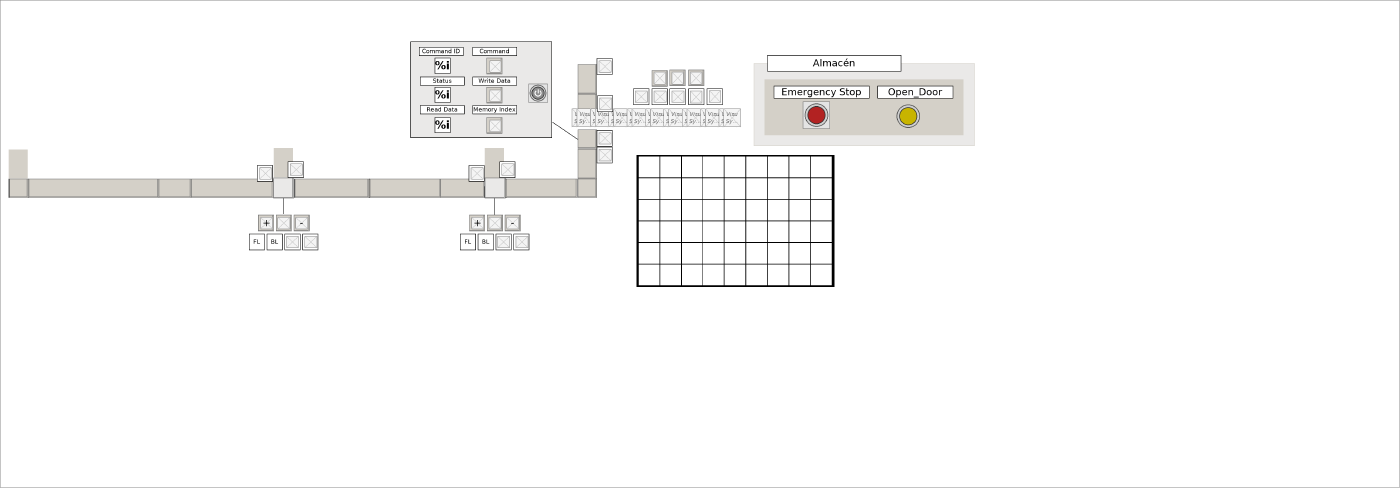
VISUALIZATION Linea_Almacen_Manual  // 2593x904
    Line (916,352) (916,399)
    Rectangle (889,284 55x35), angle 90
    Rectangle (155,228 35x241), angle 90
    Rectangle (984,282 35x132), angle 90
    Rectangle (306,318 35x60), angle 90
    Rectangle (412,272 35x152), angle 90
    Rectangle (506,329 38x38), angle 90
    Rectangle (597,280 35x137), angle 90
    Rectangle (732,283 35x131), angle 90
    Rectangle (839,308 35x81), angle 90
    Rectangle (906,336 21x38), angle 90
    Rectangle (17,331 35x35), angle 90
    Rectangle (8,286 53x35), angle 90
    Rectangle (498,284 54x35), angle 90
    Line (525,349) (525,396)
    InvisibleInput (1761,606 90x136)
    InvisibleInput (582,613 18x35)
    Button (17,331 35x35), colour toggle: GVL.Curved_Roller_Conveyor_1_CCW, pressed state: GVL.Curved_Roller_Conveyor_1_CCW
        OnMouseClick: toggle GVL.Curved_Roller_Conveyor_1_CCW
    Button (53,331 241x35), colour toggle: GVL.Roller_Conveyor_6m_1, pressed state: GVL.Roller_Conveyor_6m_1
        OnMouseClick: toggle GVL.Roller_Conveyor_6m_1
    Button (294,331 60x35), colour toggle: GVL.Chain_Transfer_1_mas, pressed state: GVL.Chain_Transfer_1_mas
        OnMouseClick: toggle GVL.Chain_Transfer_1_mas
    Button (354,331 152x35), colour toggle: GVL.Roller_Conveyor_4m_1, pressed state: GVL.Roller_Conveyor_4m_1
        OnMouseClick: toggle GVL.Roller_Conveyor_4m_1
    Button (506,329 38x38), pressed state: GVL.Roller_Conveyor_2m_2
    Button (546,331 137x35), colour toggle: GVL.Roller_Conveyor_6m_2, pressed state: GVL.Roller_Conveyor_6m_2
        OnMouseClick: toggle GVL.Roller_Conveyor_6m_2
    Button (685,331 131x35), colour toggle: GVL.Roller_Conveyor_4m_2, pressed state: GVL.Roller_Conveyor_4m_2
        OnMouseClick: toggle GVL.Roller_Conveyor_4m_2
    Button (816,331 81x35), colour toggle: GVL.Roller_Conveyor_2m_5, pressed state: GVL.Roller_Conveyor_2m_5
        OnMouseClick: toggle GVL.Roller_Conveyor_2m_5
    Button (898,329 38x38), colour toggle: GVL.Roller_Conveyor_2m_2, pressed state: GVL.Roller_Conveyor_2m_2
    Button (938,331 131x35), colour toggle: GVL.Roller_Conveyor_2m_2, pressed state: GVL.Roller_Conveyor_2m_2
        OnMouseClick: toggle GVL.Roller_Conveyor_2m_2
    Button (1070,331 35x35), colour toggle: GVL.Curved_Roller_Conveyor_2_CW, pressed state: GVL.Curved_Roller_Conveyor_2_CW
        OnMouseClick: toggle GVL.Curved_Roller_Conveyor_2_CW
    Button (1070,276 35x55), colour toggle: GVL.Roller_Conveyor_2m_8, pressed state: GVL.Roller_Conveyor_2m_8
        OnMouseClick: toggle GVL.Roller_Conveyor_2m_8
    Button (1070,240 35x35), colour toggle: GVL.Loading_Conveyor_1, pressed state: GVL.Loading_Conveyor_1
        OnMouseClick: toggle GVL.Loading_Conveyor_1
    Button (1070,174 35x35), colour toggle: GVL.Loading_Conveyor_2, pressed state: GVL.Loading_Conveyor_2
        OnMouseClick: toggle GVL.Loading_Conveyor_2
    Button (1070,119 35x55), colour toggle: GVL.Roller_Conveyor_2m_9, pressed state: GVL.Roller_Conveyor_2m_8
        OnMouseClick: toggle GVL.Roller_Conveyor_2m_9
    Rectangle (1179,287 366x244)
    Rectangle (1302,289 40x40)
    Rectangle (1302,329 40x40)
    Rectangle (1302,369 40x40)
    Rectangle (1302,409 40x40)
    Rectangle (1302,449 40x40)
    Rectangle (1302,489 40x40)
    Rectangle (1342,289 40x40)
    Rectangle (1342,329 40x40)
    Rectangle (1342,369 40x40)
    Rectangle (1342,409 40x40)
    Rectangle (1342,449 40x40)
    Rectangle (1342,489 40x40)
    Rectangle (1382,289 40x40)
    Rectangle (1382,329 40x40)
    Rectangle (1382,369 40x40)
    Rectangle (1382,409 40x40)
    Rectangle (1382,449 40x40)
    Rectangle (1382,489 40x40)
    Rectangle (1422,289 40x40)
    Rectangle (1422,329 40x40)
    Rectangle (1422,369 40x40)
    Rectangle (1422,409 40x40)
    Rectangle (1422,449 40x40)
    Rectangle (1422,489 40x40)
    Rectangle (1462,289 40x40)
    Rectangle (1462,329 40x40)
    Rectangle (1462,369 40x40)
    Rectangle (1462,409 40x40)
    Rectangle (1462,449 40x40)
    Rectangle (1462,489 40x40)
    Rectangle (1502,289 40x40)
    Rectangle (1502,329 40x40)
    Rectangle (1502,369 40x40)
    Rectangle (1502,409 40x40)
    Rectangle (1502,449 40x40)
    Rectangle (1502,489 40x40)
    Rectangle (1182,289 40x40)
    Rectangle (1182,329 40x40)
    Rectangle (1182,369 40x40)
    Rectangle (1182,409 40x40)
    Rectangle (1182,449 40x40)
    Rectangle (1182,489 40x40)
    Rectangle (1222,289 40x40)
    Rectangle (1222,329 40x40)
    Rectangle (1222,369 40x40)
    Rectangle (1222,409 40x40)
    Rectangle (1222,449 40x40)
    Rectangle (1222,489 40x40)
    Rectangle (1262,289 40x40)
    Rectangle (1262,329 40x40)
    Rectangle (1262,369 40x40)
    Rectangle (1262,409 40x40)
    Rectangle (1262,449 40x40)
    Rectangle (1262,489 40x40)
    Rectangle (1182,289 40x40), colour toggle: GVL.Clasificados[45].Visibilidad_Azul, invisible if: GVL.Clasificados[45].Visibilidad_Azul
    Rectangle (1182,329 40x40), colour toggle: GVL.Clasificados[36].Visibilidad_Azul, invisible if: GVL.Clasificados[36].Visibilidad_Azul
    Rectangle (1182,369 40x40), colour toggle: GVL.Clasificados[27].Visibilidad_Azul, invisible if: GVL.Clasificados[27].Visibilidad_Azul
    Rectangle (1182,409 40x40), colour toggle: GVL.Clasificados[18].Visibilidad_Azul, invisible if: GVL.Clasificados[18].Visibilidad_Azul
    Rectangle (1182,449 40x40), colour toggle: GVL.Clasificados[9].Visibilidad_Azul, invisible if: GVL.Clasificados[9].Visibilidad_Azul
    Rectangle (1182,489 40x40), colour toggle: GVL.Clasificados[0].Visibilidad_Azul, invisible if: GVL.Clasificados[0].Visibilidad_Azul
    Rectangle (1222,290 40x40)
    Rectangle (1222,330 40x40)
    Rectangle (1222,370 40x40)
    Rectangle (1222,410 40x40)
    Rectangle (1222,450 40x40)
    Rectangle (1222,490 40x40)
    Rectangle (1222,289 40x40), colour toggle: GVL.Clasificados[46].Visibilidad_Azul, invisible if: GVL.Clasificados[46].Visibilidad_Azul
    Rectangle (1222,329 40x40), colour toggle: GVL.Clasificados[37].Visibilidad_Azul, invisible if: GVL.Clasificados[37].Visibilidad_Azul
    Rectangle (1222,369 40x40), colour toggle: GVL.Clasificados[28].Visibilidad_Azul, invisible if: GVL.Clasificados[28].Visibilidad_Azul
    Rectangle (1222,409 40x40), colour toggle: GVL.Clasificados[19].Visibilidad_Azul, invisible if: GVL.Clasificados[19]Visibilidad_Azul
    Rectangle (1222,449 40x40), colour toggle: GVL.Clasificados[10].Visibilidad_Azul, invisible if: GVL.Clasificados[10].Visibilidad_Azul
    Rectangle (1222,489 40x40), colour toggle: GVL.Clasificados[1].Visibilidad_Azul, invisible if: GVL.Clasificados[1].Visibilidad_Azul
    Rectangle (1262,289 40x40)
    Rectangle (1262,329 40x40)
    Rectangle (1262,369 40x40)
    Rectangle (1262,409 40x40)
    Rectangle (1262,449 40x40)
    Rectangle (1262,489 40x40)
    Rectangle (1262,289 40x40), colour toggle: GVL.Clasificados[47].Visibilidad_Azul, invisible if: GVL.Clasificados[47].Visibilidad_Azul
    Rectangle (1262,329 40x40), colour toggle: GVL.Clasificados[38].Visibilidad_Azul, invisible if: GVL.Clasificados[38].Visibilidad_Azul
    Rectangle (1262,369 40x40), colour toggle: GVL.Clasificados[29].Visibilidad_Azul, invisible if: GVL.Clasificados[29].Visibilidad_Azul
    Rectangle (1262,409 40x40), colour toggle: GVL.Clasificados[20].Visibilidad_Azul, invisible if: GVL.Clasificados[20].Visibilidad_Azul
    Rectangle (1262,449 40x40), colour toggle: GVL.Clasificados[11].Visibilidad_Azul, invisible if: GVL.Clasificados[11].Visibilidad_Azul
    Rectangle (1262,489 40x40), colour toggle: GVL.Clasificados[2].Visibilidad_Azul, invisible if: GVL.Clasificados[2].Visibilidad_Azul
    Rectangle (1301,289 40x40)
    Rectangle (1301,329 40x40)
    Rectangle (1301,369 40x40)
    Rectangle (1301,409 40x40)
    Rectangle (1301,449 40x40)
    Rectangle (1301,489 40x40)
    Rectangle (1341,289 40x40)
    Rectangle (1341,329 40x40)
    Rectangle (1341,369 40x40)
    Rectangle (1341,409 40x40)
    Rectangle (1341,449 40x40)
    Rectangle (1341,489 40x40)
    Rectangle (1381,289 40x40)
    Rectangle (1381,329 40x40)
    Rectangle (1381,369 40x40)
    Rectangle (1381,409 40x40)
    Rectangle (1381,449 40x40)
    Rectangle (1381,489 40x40)
    Rectangle (1301,289 40x40), colour toggle: GVL.Clasificados[48].Visibilidad_Azul, invisible if: GVL.Clasificados[48].Visibilidad_Azul
    Rectangle (1301,329 40x40), colour toggle: GVL.Clasificados[39].Visibilidad_Azul, invisible if: GVL.Clasificados[39].Visibilidad_Azul
    Rectangle (1301,369 40x40), colour toggle: GVL.Clasificados[30].Visibilidad_Azul, invisible if: GVL.Clasificados[30].Visibilidad_Azul
    Rectangle (1301,409 40x40), colour toggle: GVL.Clasificados[21].Visibilidad_Azul, invisible if: GVL.Clasificados[21].Visibilidad_Azul
    Rectangle (1301,449 40x40), colour toggle: GVL.Clasificados[12].Visibilidad_Azul, invisible if: GVL.Clasificados[12].Visibilidad_Azul
    Rectangle (1301,489 40x40), colour toggle: GVL.Clasificados[3].Visibilidad_Azul, invisible if: GVL.Clasificados[3].Visibilidad_Azul
    Rectangle (1341,290 40x40)
    Rectangle (1341,330 40x40)
    Rectangle (1341,370 40x40)
    Rectangle (1341,410 40x40)
    Rectangle (1341,450 40x40)
    Rectangle (1341,490 40x40)
    Rectangle (1341,289 40x40), colour toggle: GVL.Clasificados[49].Visibilidad_Azul, invisible if: GVL.Clasificados[49].Visibilidad_Azul
    Rectangle (1341,329 40x40), colour toggle: GVL.Clasificados[40].Visibilidad_Azul, invisible if: GVL.Clasificados[40].Visibilidad_Azul
    Rectangle (1341,369 40x40), colour toggle: GVL.Clasificados[31].Visibilidad_Azul, invisible if: GVL.Clasificados[31].Visibilidad_Azul
    Rectangle (1341,409 40x40), colour toggle: GVL.Clasificados[22].Visibilidad_Azul, invisible if: GVL.Clasificados[22].Visibilidad_Azul
    Rectangle (1341,449 40x40), colour toggle: GVL.Clasificados[13].Visibilidad_Azul, invisible if: GVL.Clasificados[13].Visibilidad_Azul
    Rectangle (1341,489 40x40), colour toggle: GVL.Clasificados[4].Visibilidad_Azul, invisible if: GVL.Clasificados[4].Visibilidad_Azul
    Rectangle (1381,289 40x40)
    Rectangle (1381,329 40x40)
    Rectangle (1381,369 40x40)
    Rectangle (1381,409 40x40)
    Rectangle (1381,449 40x40)
    Rectangle (1381,489 40x40)
    Rectangle (1381,289 40x40), colour toggle: GVL.Clasificados[50].Visibilidad_Azul, invisible if: GVL.Clasificados[50].Visibilidad_Azul
    Rectangle (1381,329 40x40), colour toggle: GVL.Clasificados[41].Visibilidad_Azul, invisible if: GVL.Clasificados[41].Visibilidad_Azul
    Rectangle (1381,369 40x40), colour toggle: GVL.Clasificados[32].Visibilidad_Azul, invisible if: GVL.Clasificados[32].Visibilidad_Azul
    Rectangle (1381,409 40x40), colour toggle: GVL.Clasificados[23].Visibilidad_Azul, invisible if: GVL.Clasificados[23].Visibilidad_Azul
    Rectangle (1381,449 40x40), colour toggle: GVL.Clasificados[14].Visibilidad_Azul, invisible if: GVL.Clasificados[14].Visibilidad_Azul
    Rectangle (1381,489 40x40), colour toggle: GVL.Clasificados[5].Visibilidad_Azul, invisible if: GVL.Clasificados[5].Visibilidad_Azul
    Rectangle (1421,289 40x40)
    Rectangle (1421,329 40x40)
    Rectangle (1421,369 40x40)
    Rectangle (1421,409 40x40)
    Rectangle (1421,449 40x40)
    Rectangle (1421,489 40x40)
    Rectangle (1461,289 40x40)
    Rectangle (1461,329 40x40)
    Rectangle (1461,369 40x40)
    Rectangle (1461,409 40x40)
    Rectangle (1461,449 40x40)
    Rectangle (1461,489 40x40)
    Rectangle (1501,289 40x40)
    Rectangle (1501,329 40x40)
    Rectangle (1501,369 40x40)
    Rectangle (1501,409 40x40)
    Rectangle (1501,449 40x40)
    Rectangle (1501,489 40x40)
    Rectangle (1421,289 40x40), colour toggle: GVL.Clasificados[51].Visibilidad_Azul, invisible if: GVL.Clasificados[51].Visibilidad_Azul
    Rectangle (1421,329 40x40), colour toggle: GVL.Clasificados[42].Visibilidad_Azul, invisible if: GVL.Clasificados[42].Visibilidad_Azul
    Rectangle (1421,369 40x40), colour toggle: GVL.Clasificados[33].Visibilidad_Azul, invisible if: GVL.Clasificados[33].Visibilidad_Azul
    Rectangle (1421,409 40x40), colour toggle: GVL.Clasificados[24].Visibilidad_Azul, invisible if: GVL.Clasificados[24].Visibilidad_Azul
    Rectangle (1421,449 40x40), colour toggle: GVL.Clasificados[15].Visibilidad_Azul, invisible if: GVL.Clasificados[15].Visibilidad_Azul
    Rectangle (1421,489 40x40), colour toggle: GVL.Clasificados[6].Visibilidad_Azul, invisible if: GVL.Clasificados[6].Visibilidad_Azul
    Rectangle (1461,290 40x40)
    Rectangle (1461,330 40x40)
    Rectangle (1461,370 40x40)
    Rectangle (1461,410 40x40)
    Rectangle (1461,450 40x40)
    Rectangle (1461,490 40x40)
    Rectangle (1461,289 40x40), colour toggle: GVL.Clasificados[52].Visibilidad_Azul, invisible if: GVL.Clasificados[52].Visibilidad_Azul
    Rectangle (1461,329 40x40), colour toggle: GVL.Clasificados[43].Visibilidad_Azul, invisible if: GVL.Clasificados[43].Visibilidad_Azul
    Rectangle (1461,369 40x40), colour toggle: GVL.Clasificados[34].Visibilidad_Azul, invisible if: GVL.Clasificados[34].Visibilidad_Azul
    Rectangle (1461,409 40x40), colour toggle: GVL.Clasificados[25].Visibilidad_Azul, invisible if: GVL.Clasificados[25].Visibilidad_Azul
    Rectangle (1461,449 40x40), colour toggle: GVL.Clasificados[16].Visibilidad_Azul, invisible if: GVL.Clasificados[16].Visibilidad_Azul
    Rectangle (1461,489 40x40), colour toggle: GVL.Clasificados[7].Visibilidad_Azul, invisible if: GVL.Clasificados[7].Visibilidad_Azul
    Rectangle (1501,289 40x40)
    Rectangle (1501,329 40x40)
    Rectangle (1501,369 40x40)
    Rectangle (1501,409 40x40)
    Rectangle (1501,449 40x40)
    Rectangle (1501,489 40x40)
    Rectangle (1501,289 40x40), colour toggle: GVL.Clasificados[53].Visibilidad_Azul, invisible if: GVL.Clasificados[53].Visibilidad_Azul
    Rectangle (1501,329 40x40), colour toggle: GVL.Clasificados[44].Visibilidad_Azul, invisible if: GVL.Clasificados[44].Visibilidad_Azul
    Rectangle (1501,369 40x40), colour toggle: GVL.Clasificados[35].Visibilidad_Azul, invisible if: GVL.Clasificados[35].Visibilidad_Azul
    Rectangle (1501,409 40x40), colour toggle: GVL.Clasificados[26].Visibilidad_Azul, invisible if: GVL.Clasificados[26].Visibilidad_Azul
    Rectangle (1501,449 40x40), colour toggle: GVL.Clasificados[17].Visibilidad_Azul, invisible if: GVL.Clasificados[17].Visibilidad_Azul
    Rectangle (1501,489 40x40), colour toggle: GVL.Clasificados[8].Visibilidad_Azul, invisible if: GVL.Clasificados[8].Visibilidad_Azul
    Rectangle (1182,289 40x40), colour toggle: GVL.Clasificados[45].Visibilidad_Verde, invisible if: GVL.Clasificados[45].Visibilidad_Verde
    Rectangle (1182,329 40x40), colour toggle: GVL.Clasificados[36].Visibilidad_Verde, invisible if: GVL.Clasificados[36].Visibilidad_Verde
    Rectangle (1182,369 40x40), colour toggle: GVL.Clasificados[27].Visibilidad_Verde, invisible if: GVL.Clasificados[27].Visibilidad_Verde
    Rectangle (1182,409 40x40), colour toggle: GVL.Clasificados[18].Visibilidad_Verde, invisible if: GVL.Clasificados[18].Visibilidad_Verde
    Rectangle (1182,449 40x40), colour toggle: GVL.Clasificados[9].Visibilidad_Verde, invisible if: GVL.Clasificados[9].Visibilidad_Verde
    Rectangle (1182,489 40x40), colour toggle: GVL.Clasificados[0].Visibilidad_Verde, invisible if: GVL.Clasificados[0].Visibilidad_Verde
    Rectangle (1222,289 40x40), colour toggle: GVL.Clasificados[46].Visibilidad_Verde, invisible if: GVL.Clasificados[46].Visibilidad_Verde
    Rectangle (1222,329 40x40), colour toggle: GVL.Clasificados[37].Visibilidad_Verde, invisible if: GVL.Clasificados[37].Visibilidad_Verde
    Rectangle (1222,369 40x40), colour toggle: GVL.Clasificados[28].Visibilidad_Verde, invisible if: GVL.Clasificados[28].Visibilidad_Verde
    Rectangle (1222,409 40x40), colour toggle: GVL.Clasificados[19].Visibilidad_Verde, invisible if: GVL.Clasificados[19].Visibilidad_Verde
    Rectangle (1222,449 40x40), colour toggle: GVL.Clasificados[10].Visibilidad_Verde, invisible if: GVL.Clasificados[10].Visibilidad_Verde
    Rectangle (1222,489 40x40), colour toggle: GVL.Clasificados[1].Visibilidad_Verde, invisible if: GVL.Clasificados[1].Visibilidad_Verde
    Rectangle (1262,289 40x40), colour toggle: GVL.Clasificados[47].Visibilidad_Verde, invisible if: GVL.Clasificados[47].Visibilidad_Verde
    Rectangle (1262,329 40x40), colour toggle: GVL.Clasificados[38].Visibilidad_Verde, invisible if: GVL.Clasificados[38].Visibilidad_Verde
    Rectangle (1262,369 40x40), colour toggle: GVL.Clasificados[29].Visibilidad_Verde, invisible if: GVL.Clasificados[29].Visibilidad_Verde
    Rectangle (1262,409 40x40), colour toggle: GVL.Clasificados[20].Visibilidad_Verde, invisible if: GVL.Clasificados[20].Visibilidad_Verde
    Rectangle (1262,449 40x40), colour toggle: GVL.Clasificados[11].Visibilidad_Verde, invisible if: GVL.Clasificados[11].Visibilidad_Verde
    Rectangle (1262,489 40x40), colour toggle: GVL.Clasificados[2].Visibilidad_Verde, invisible if: GVL.Clasificados[2].Visibilidad_Verde
    Rectangle (1301,289 40x40), colour toggle: GVL.Clasificados[48].Visibilidad_Verde, invisible if: GVL.Clasificados[48].Visibilidad_Verde
    Rectangle (1301,329 40x40), colour toggle: GVL.Clasificados[39].Visibilidad_Verde, invisible if: GVL.Clasificados[39].Visibilidad_Verde
    Rectangle (1301,369 40x40), colour toggle: GVL.Clasificados[30].Visibilidad_Verde, invisible if: GVL.Clasificados[30].Visibilidad_Verde
    Rectangle (1301,409 40x40), colour toggle: GVL.Clasificados[21].Visibilidad_Verde, invisible if: GVL.Clasificados[21].Visibilidad_Verde
    Rectangle (1301,449 40x40), colour toggle: GVL.Clasificados[12].Visibilidad_Verde, invisible if: GVL.Clasificados[12].Visibilidad_Verde
    Rectangle (1301,489 40x40), colour toggle: GVL.Clasificados[3].Visibilidad_Verde, invisible if: GVL.Clasificados[3].Visibilidad_Verde
    Rectangle (1341,289 40x40), colour toggle: GVL.Clasificados[49].Visibilidad_Verde, invisible if: GVL.Clasificados[49].Visibilidad_Verde
    Rectangle (1341,329 40x40), colour toggle: GVL.Clasificados[40].Visibilidad_Verde, invisible if: GVL.Clasificados[40].Visibilidad_Verde
    Rectangle (1341,369 40x40), colour toggle: GVL.Clasificados[31].Visibilidad_Verde, invisible if: GVL.Clasificados[31].Visibilidad_Verde
    Rectangle (1341,409 40x40), colour toggle: GVL.Clasificados[22].Visibilidad_Verde, invisible if: GVL.Clasificados[22].Visibilidad_Verde
    Rectangle (1341,449 40x40), colour toggle: GVL.Clasificados[13].Visibilidad_Verde, invisible if: GVL.Clasificados[13].Visibilidad_Verde
    Rectangle (1341,489 40x40), colour toggle: GVL.Clasificados[4].Visibilidad_Verde, invisible if: GVL.Clasificados[4].Visibilidad_Verde
    Rectangle (1381,289 40x40), colour toggle: GVL.Clasificados[50].Visibilidad_Verde, invisible if: GVL.Clasificados[50].Visibilidad_Verde
    Rectangle (1381,329 40x40), colour toggle: GVL.Clasificados[41].Visibilidad_Verde, invisible if: GVL.Clasificados[41].Visibilidad_Verde
    Rectangle (1381,369 40x40), colour toggle: GVL.Clasificados[32].Visibilidad_Verde, invisible if: GVL.Clasificados[32].Visibilidad_Verde
    Rectangle (1381,409 40x40), colour toggle: GVL.Clasificados[23].Visibilidad_Verde, invisible if: GVL.Clasificados[23].Visibilidad_Verde
    Rectangle (1381,449 40x40), colour toggle: GVL.Clasificados[14].Visibilidad_Verde, invisible if: GVL.Clasificados[14].Visibilidad_Verde
    Rectangle (1381,489 40x40), colour toggle: GVL.Clasificados[5].Visibilidad_Verde, invisible if: GVL.Clasificados[5].Visibilidad_Verde
    Rectangle (1421,289 40x40), colour toggle: GVL.Clasificados[51].Visibilidad_Verde, invisible if: GVL.Clasificados[51].Visibilidad_Verde
    Rectangle (1421,329 40x40), colour toggle: GVL.Clasificados[42].Visibilidad_Verde, invisible if: GVL.Clasificados[42].Visibilidad_Verde
    Rectangle (1421,369 40x40), colour toggle: GVL.Clasificados[33].Visibilidad_Verde, invisible if: GVL.Clasificados[33].Visibilidad_Verde
    Rectangle (1421,409 40x40), colour toggle: GVL.Clasificados[24].Visibilidad_Verde, invisible if: GVL.Clasificados[24].Visibilidad_Verde
    Rectangle (1421,449 40x40), colour toggle: GVL.Clasificados[15].Visibilidad_Verde, invisible if: GVL.Clasificados[15].Visibilidad_Verde
    Rectangle (1421,489 40x40), colour toggle: GVL.Clasificados[6].Visibilidad_Verde, invisible if: GVL.Clasificados[6].Visibilidad_Verde
    Rectangle (1461,289 40x40), colour toggle: GVL.Clasificados[52].Visibilidad_Verde, invisible if: GVL.Clasificados[52].Visibilidad_Verde
    Rectangle (1461,329 40x40), colour toggle: GVL.Clasificados[43].Visibilidad_Verde, invisible if: GVL.Clasificados[43].Visibilidad_Verde
    Rectangle (1461,369 40x40), colour toggle: GVL.Clasificados[34].Visibilidad_Verde, invisible if: GVL.Clasificados[34].Visibilidad_Verde
    Rectangle (1461,409 40x40), colour toggle: GVL.Clasificados[25].Visibilidad_Verde, invisible if: GVL.Clasificados[25].Visibilidad_Verde
    Rectangle (1461,449 40x40), colour toggle: GVL.Clasificados[16].Visibilidad_Verde, invisible if: GVL.Clasificados[16].Visibilidad_Verde
    Rectangle (1461,489 40x40), colour toggle: GVL.Clasificados[7].Visibilidad_Verde, invisible if: GVL.Clasificados[7].Visibilidad_Verde
    Rectangle (1501,289 40x40), colour toggle: GVL.Clasificados[53].Visibilidad_Verde, invisible if: GVL.Clasificados[53].Visibilidad_Verde
    Rectangle (1501,329 40x40), colour toggle: GVL.Clasificados[44].Visibilidad_Verde, invisible if: GVL.Clasificados[44].Visibilidad_Verde
    Rectangle (1501,369 40x40), colour toggle: GVL.Clasificados[35].Visibilidad_Verde, invisible if: GVL.Clasificados[35].Visibilidad_Verde
    Rectangle (1501,409 40x40), colour toggle: GVL.Clasificados[26].Visibilidad_Verde, invisible if: GVL.Clasificados[26].Visibilidad_Verde
    Rectangle (1501,449 40x40), colour toggle: GVL.Clasificados[17].Visibilidad_Verde, invisible if: GVL.Clasificados[17].Visibilidad_Verde
    Rectangle (1501,489 40x40), colour toggle: GVL.Clasificados[8].Visibilidad_Verde, invisible if: GVL.Clasificados[8].Visibilidad_Verde
    Rectangle (1421,289 40x40), colour toggle: GVL.Clasificados[51].Visibilidad_Metal, invisible if: GVL.Clasificados[51].Visibilidad_Metal
    Rectangle (1421,369 40x40), colour toggle: GVL.Clasificados[33].Visibilidad_Metal, invisible if: GVL.Clasificados[33].Visibilidad_Metal
    Rectangle (1421,329 40x40), colour toggle: GVL.Clasificados[42].Visibilidad_Metal, invisible if: GVL.Clasificados[42].Visibilidad_Metal
    Rectangle (1421,409 40x40), colour toggle: GVL.Clasificados[24].Visibilidad_Metal, invisible if: GVL.Clasificados[24].Visibilidad_Metal
    Rectangle (1421,449 40x40), colour toggle: GVL.Clasificados[15].Visibilidad_Metal, invisible if: GVL.Clasificados[15].Visibilidad_Metal
    Rectangle (1421,489 40x40), colour toggle: GVL.Clasificados[6].Visibilidad_Metal, invisible if: GVL.Clasificados[6].Visibilidad_Metal
    Rectangle (1461,289 40x40), colour toggle: GVL.Clasificados[52].Visibilidad_Metal, invisible if: GVL.Clasificados[52].Visibilidad_Metal
    Rectangle (1461,369 40x40), colour toggle: GVL.Clasificados[34].Visibilidad_Metal, invisible if: GVL.Clasificados[34].Visibilidad_Metal
    Rectangle (1461,329 40x40), colour toggle: GVL.Clasificados[43].Visibilidad_Metal, invisible if: GVL.Clasificados[43].Visibilidad_Metal
    Rectangle (1461,409 40x40), colour toggle: GVL.Clasificados[25].Visibilidad_Metal, invisible if: GVL.Clasificados[25].Visibilidad_Metal
    Rectangle (1461,449 40x40), colour toggle: GVL.Clasificados[16].Visibilidad_Metal, invisible if: GVL.Clasificados[16].Visibilidad_Metal
    Rectangle (1461,489 40x40), colour toggle: GVL.Clasificados[7].Visibilidad_Metal, invisible if: GVL.Clasificados[7].Visibilidad_Metal
    Rectangle (1501,289 40x40), colour toggle: GVL.Clasificados[53].Visibilidad_Metal, invisible if: GVL.Clasificados[53].Visibilidad_Metal
    Rectangle (1501,369 40x40), colour toggle: GVL.Clasificados[35].Visibilidad_Metal, invisible if: GVL.Clasificados[35].Visibilidad_Metal
    Rectangle (1501,329 40x40), colour toggle: GVL.Clasificados[44].Visibilidad_Metal, invisible if: GVL.Clasificados[44].Visibilidad_Metal
    Rectangle (1501,409 40x40), colour toggle: GVL.Clasificados[26].Visibilidad_Metal, invisible if: GVL.Clasificados[26].Visibilidad_Metal
    Rectangle (1501,449 40x40), colour toggle: GVL.Clasificados[17].Visibilidad_Metal, invisible if: GVL.Clasificados[17].Visibilidad_Metal
    Rectangle (1501,489 40x40), colour toggle: GVL.Clasificados[8].Visibilidad_Metal, invisible if: GVL.Clasificados[8].Visibilidad_Metal
    Rectangle (1182,289 40x40), colour toggle: GVL.Clasificados[45].Visibilidad_Metal, invisible if: GVL.Clasificados[45].Visibilidad_Metal
    Rectangle (1182,369 40x40), colour toggle: GVL.Clasificados[27].Visibilidad_Metal, invisible if: GVL.Clasificados[27].Visibilidad_Metal
    Rectangle (1182,329 40x40), colour toggle: GVL.Clasificados[36].Visibilidad_Metal, invisible if: GVL.Clasificados[36].Visibilidad_Metal
    Rectangle (1182,409 40x40), colour toggle: GVL.Clasificados[18].Visibilidad_Metal, invisible if: GVL.Clasificados[18].Visibilidad_Metal
    Rectangle (1182,449 40x40), colour toggle: GVL.Clasificados[9].Visibilidad_Metal, invisible if: GVL.Clasificados[9].Visibilidad_Metal
    Rectangle (1182,489 40x40), colour toggle: GVL.Clasificados[0].Visibilidad_Metal, invisible if: GVL.Clasificados[0].Visibilidad_Metal
    Rectangle (1222,289 40x40), colour toggle: GVL.Clasificados[46].Visibilidad_Metal, invisible if: GVL.Clasificados[46].Visibilidad_Metal
    Rectangle (1222,369 40x40), colour toggle: GVL.Clasificados[28].Visibilidad_Metal, invisible if: GVL.Clasificados[28].Visibilidad_Metal
    Rectangle (1222,329 40x40), colour toggle: GVL.Clasificados[37].Visibilidad_Metal, invisible if: GVL.Clasificados[37].Visibilidad_Metal
    Rectangle (1222,409 40x40), colour toggle: GVL.Clasificados[19].Visibilidad_Metal, invisible if: GVL.Clasificados[19].Visibilidad_Metal
    Rectangle (1222,449 40x40), colour toggle: GVL.Clasificados[10].Visibilidad_Metal, invisible if: GVL.Clasificados[10].Visibilidad_Metal
    Rectangle (1222,489 40x40), colour toggle: GVL.Clasificados[1].Visibilidad_Metal, invisible if: GVL.Clasificados[1].Visibilidad_Metal
    Rectangle (1262,289 40x40), colour toggle: GVL.Clasificados[47].Visibilidad_Metal, invisible if: GVL.Clasificados[47].Visibilidad_Metal
    Rectangle (1262,369 40x40), colour toggle: GVL.Clasificados[29].Visibilidad_Metal, invisible if: GVL.Clasificados[29].Visibilidad_Metal
    Rectangle (1262,329 40x40), colour toggle: GVL.Clasificados[38].Visibilidad_Metal, invisible if: GVL.Clasificados[38].Visibilidad_Metal
    Rectangle (1262,409 40x40), colour toggle: GVL.Clasificados[20].Visibilidad_Metal, invisible if: GVL.Clasificados[20].Visibilidad_Metal
    Rectangle (1262,449 40x40), colour toggle: GVL.Clasificados[11].Visibilidad_Metal, invisible if: GVL.Clasificados[11].Visibilidad_Metal
    Rectangle (1262,489 40x40), colour toggle: GVL.Clasificados[2].Visibilidad_Metal, invisible if: GVL.Clasificados[2].Visibilidad_Metal
    Rectangle (1302,289 40x40), colour toggle: GVL.Clasificados[48].Visibilidad_Metal, invisible if: GVL.Clasificados[48].Visibilidad_Metal
    Rectangle (1302,369 40x40), colour toggle: GVL.Clasificados[30].Visibilidad_Metal, invisible if: GVL.Clasificados[30].Visibilidad_Metal
    Rectangle (1302,329 40x40), colour toggle: GVL.Clasificados[39].Visibilidad_Metal, invisible if: GVL.Clasificados[39].Visibilidad_Metal
    Rectangle (1302,409 40x40), colour toggle: GVL.Clasificados[21].Visibilidad_Metal, invisible if: GVL.Clasificados[21].Visibilidad_Metal
    Rectangle (1302,449 40x40), colour toggle: GVL.Clasificados[12].Visibilidad_Metal, invisible if: GVL.Clasificados[12].Visibilidad_Metal
    Rectangle (1302,489 40x40), colour toggle: GVL.Clasificados[3].Visibilidad_Metal, invisible if: GVL.Clasificados[3].Visibilidad_Metal
    Rectangle (1341,289 40x40), colour toggle: GVL.Clasificados[49].Visibilidad_Metal, invisible if: GVL.Clasificados[49 ].Visibilidad_Metal
    Rectangle (1341,369 40x40), colour toggle: GVL.Clasificados[31].Visibilidad_Metal, invisible if: GVL.Clasificados[31].Visibilidad_Metal
    Rectangle (1341,329 40x40), colour toggle: GVL.Clasificados[40].Visibilidad_Metal, invisible if: GVL.Clasificados[40].Visibilidad_Metal
    Rectangle (1341,409 40x40), colour toggle: GVL.Clasificados[22].Visibilidad_Metal, invisible if: GVL.Clasificados[22].Visibilidad_Metal
    Rectangle (1341,449 40x40), colour toggle: GVL.Clasificados[13].Visibilidad_Metal, invisible if: GVL.Clasificados[13].Visibilidad_Metal
    Rectangle (1341,489 40x40), colour toggle: GVL.Clasificados[4].Visibilidad_Metal, invisible if: GVL.Clasificados[4].Visibilidad_Metal
    Rectangle (1381,289 40x40), colour toggle: GVL.Clasificados[50].Visibilidad_Metal, invisible if: GVL.Clasificados[50].Visibilidad_Metal
    Rectangle (1381,369 40x40), colour toggle: GVL.Clasificados[32].Visibilidad_Metal, invisible if: GVL.Clasificados[32].Visibilidad_Metal
    Rectangle (1381,329 40x40), colour toggle: GVL.Clasificados[41].Visibilidad_Metal, invisible if: GVL.Clasificados[41].Visibilidad_Metal
    Rectangle (1381,409 40x40), colour toggle: GVL.Clasificados[23].Visibilidad_Metal, invisible if: GVL.Clasificados[23].Visibilidad_Metal
    Rectangle (1381,449 40x40), colour toggle: GVL.Clasificados[14].Visibilidad_Metal, invisible if: GVL.Clasificados[14].Visibilidad_Metal
    Rectangle (1381,489 40x40), colour toggle: GVL.Clasificados[5].Visibilidad_Metal, invisible if: GVL.Clasificados[5].Visibilidad_Metal
    Rectangle (1182,289 40x40), invisible if: GVL.Clasificados[45].Visibilidad_Vacio
    Rectangle (1182,329 40x40), invisible if: GVL.Clasificados[36].Visibilidad_Vacio
    Rectangle (1182,369 40x40), invisible if: GVL.Clasificados[27].Visibilidad_Vacio
    Rectangle (1182,409 40x40), invisible if: GVL.Clasificados[18].Visibilidad_Vacio
    Rectangle (1182,449 40x40), invisible if: GVL.Clasificados[9].Visibilidad_Vacio
    Rectangle (1182,489 40x40), invisible if: GVL.Clasificados[0].Visibilidad_Vacio
    Rectangle (1222,289 40x40), invisible if: GVL.Clasificados[46].Visibilidad_Vacio
    Rectangle (1222,329 40x40), invisible if: GVL.Clasificados[37].Visibilidad_Vacio
    Rectangle (1222,369 40x40), invisible if: GVL.Clasificados[28].Visibilidad_Vacio
    Rectangle (1222,409 40x40), invisible if: GVL.Clasificados[19].Visibilidad_Vacio
    Rectangle (1222,449 40x40), invisible if: GVL.Clasificados[10].Visibilidad_Vacio
    Rectangle (1222,489 40x40), invisible if: GVL.Clasificados[1].Visibilidad_Vacio
    Rectangle (1262,289 40x40), invisible if: GVL.Clasificados[47].Visibilidad_Vacio
    Rectangle (1262,329 40x40), invisible if: GVL.Clasificados[38].Visibilidad_Vacio
    Rectangle (1262,369 40x40), invisible if: GVL.Clasificados[29].Visibilidad_Vacio
    Rectangle (1262,409 40x40), invisible if: GVL.Clasificados[20].Visibilidad_Vacio
    Rectangle (1262,449 40x40), invisible if: GVL.Clasificados[11].Visibilidad_Vacio
    Rectangle (1262,489 40x40), invisible if: GVL.Clasificados[2].Visibilidad_Vacio
    Rectangle (1301,289 40x40), invisible if: GVL.Clasificados[48].Visibilidad_Vacio
    Rectangle (1301,329 40x40), invisible if: GVL.Clasificados[39].Visibilidad_Vacio
    Rectangle (1301,369 40x40), invisible if: GVL.Clasificados[30].Visibilidad_Vacio
    Rectangle (1301,409 40x40), invisible if: GVL.Clasificados[21].Visibilidad_Vacio
    Rectangle (1301,449 40x40), invisible if: GVL.Clasificados[12].Visibilidad_Vacio
    Rectangle (1301,489 40x40), invisible if: GVL.Clasificados[3].Visibilidad_Vacio
    Rectangle (1341,289 40x40), invisible if: GVL.Clasificados[49].Visibilidad_Vacio
    Rectangle (1341,329 40x40), invisible if: GVL.Clasificados[40].Visibilidad_Vacio
    Rectangle (1341,369 40x40), invisible if: GVL.Clasificados[31].Visibilidad_Vacio
    Rectangle (1341,409 40x40), invisible if: GVL.Clasificados[22].Visibilidad_Vacio
    Rectangle (1341,449 40x40), invisible if: GVL.Clasificados[13].Visibilidad_Vacio
    Rectangle (1341,489 40x40), invisible if: GVL.Clasificados[4].Visibilidad_Vacio
    Rectangle (1381,289 40x40), invisible if: GVL.Clasificados[50].Visibilidad_Vacio
    Rectangle (1381,329 40x40), invisible if: GVL.Clasificados[41].Visibilidad_Vacio
    Rectangle (1381,369 40x40), invisible if: GVL.Clasificados[32].Visibilidad_Vacio
    Rectangle (1381,409 40x40), invisible if: GVL.Clasificados[23].Visibilidad_Vacio
    Rectangle (1381,449 40x40), invisible if: GVL.Clasificados[14].Visibilidad_Vacio
    Rectangle (1381,489 40x40), invisible if: GVL.Clasificados[5].Visibilidad_Vacio
    Rectangle (1421,289 40x40), invisible if: GVL.Clasificados[51].Visibilidad_Vacio
    Rectangle (1421,329 40x40), invisible if: GVL.Clasificados[42].Visibilidad_Vacio
    Rectangle (1421,369 40x40), invisible if: GVL.Clasificados[33].Visibilidad_Vacio
    Rectangle (1421,409 40x40), invisible if: GVL.Clasificados[24].Visibilidad_Vacio
    Rectangle (1421,449 40x40), invisible if: GVL.Clasificados[15].Visibilidad_Vacio
    Rectangle (1421,489 40x40), invisible if: GVL.Clasificados[6].Visibilidad_Vacio
    Rectangle (1461,289 40x40), invisible if: GVL.Clasificados[52].Visibilidad_Vacio
    Rectangle (1461,329 40x40), invisible if: GVL.Clasificados[43].Visibilidad_Vacio
    Rectangle (1461,369 40x40), invisible if: GVL.Clasificados[34].Visibilidad_Vacio
    Rectangle (1461,409 40x40), invisible if: GVL.Clasificados[25].Visibilidad_Vacio
    Rectangle (1461,449 40x40), invisible if: GVL.Clasificados[16].Visibilidad_Vacio
    Rectangle (1461,489 40x40), invisible if: GVL.Clasificados[7].Visibilidad_Vacio
    Rectangle (1501,289 40x40), invisible if: GVL.Clasificados[53].Visibilidad_Vacio
    Rectangle (1501,329 40x40), invisible if: GVL.Clasificados[44].Visibilidad_Vacio
    Rectangle (1501,369 40x40), invisible if: GVL.Clasificados[35].Visibilidad_Vacio
    Rectangle (1501,409 40x40), invisible if: GVL.Clasificados[26].Visibilidad_Vacio
    Rectangle (1501,449 40x40), invisible if: GVL.Clasificados[17].Visibilidad_Vacio
    Rectangle (1501,489 40x40), invisible if: GVL.Clasificados[8].Visibilidad_Vacio
    Group (1059,201 330x48)
        Group (0,0 126x48)
            Group (0,0 92x48)
                Group (0,0 58x48)
                    Rectangle (8,5 24x23)
                    Image (0,0 32x34), image: VisuSymbols.Symbols.ArrowForward
                    Image (9,0 32x34), angle 90, image: VisuSymbols.Symbols.ArrowDown
                Group (34,0 58x48)
                    Rectangle (8,5 24x23)
                    Image (0,0 32x34), image: VisuSymbols.Symbols.ArrowForward
                    Image (9,0 32x34), angle 90, image: VisuSymbols.Symbols.ArrowDown
            Group (68,0 58x48)
                Rectangle (8,5 24x23)
                Image (0,0 32x34), image: VisuSymbols.Symbols.ArrowForward
                Image (9,0 32x34), angle 90, image: VisuSymbols.Symbols.ArrowDown
        Group (102,0 126x48)
            Group (0,0 92x48)
                Group (0,0 58x48)
                    Rectangle (8,5 24x23)
                    Image (0,0 32x34), image: VisuSymbols.Symbols.ArrowForward
                    Image (9,0 32x34), angle 90, image: VisuSymbols.Symbols.ArrowDown
                Group (34,0 58x48)
                    Rectangle (8,5 24x23)
                    Image (0,0 32x34), image: VisuSymbols.Symbols.ArrowForward
                    Image (9,0 32x34), angle 90, image: VisuSymbols.Symbols.ArrowDown
            Group (68,0 58x48)
                Rectangle (8,5 24x23)
                Image (0,0 32x34), image: VisuSymbols.Symbols.ArrowForward
                Image (9,0 32x34), angle 90, image: VisuSymbols.Symbols.ArrowDown
        Group (204,0 126x48)
            Group (0,0 92x48)
                Group (0,0 58x48)
                    Rectangle (8,5 24x23)
                    Image (0,0 32x34), image: VisuSymbols.Symbols.ArrowForward
                    Image (9,0 32x34), angle 90, image: VisuSymbols.Symbols.ArrowDown
                Group (34,0 58x48)
                    Rectangle (8,5 24x23)
                    Image (0,0 32x34), image: VisuSymbols.Symbols.ArrowForward
                    Image (9,0 32x34), angle 90, image: VisuSymbols.Symbols.ArrowDown
            Group (68,0 58x48)
                Rectangle (8,5 24x23)
                Image (0,0 32x34), image: VisuSymbols.Symbols.ArrowForward
                Image (9,0 32x34), angle 90, image: VisuSymbols.Symbols.ArrowDown
    Group (476,306 29x30), colour toggle: GVL.Diffuse_Sensor_39
        RoundedRectangle (0,0 29x30), colour toggle: GVL.Diffuse_Sensor_4
        Image (4,4 23x22), image: VisuSymbols.Symbols.RSS1
    Group (533,299 29x30), colour toggle: GVL.Diffuse_Sensor_40
        RoundedRectangle (0,0 29x30), colour toggle: GVL.Diffuse_Sensor_4
        Image (4,4 23x22), image: VisuSymbols.Symbols.RSS1
    Group (868,306 29x30), colour toggle: GVL.Diffuse_Sensor_41
        RoundedRectangle (0,0 29x30), colour toggle: GVL.Diffuse_Sensor_4
        Image (4,4 23x22), image: VisuSymbols.Symbols.RSS1
    Group (925,299 29x30), colour toggle: GVL.Diffuse_Sensor_42
        RoundedRectangle (0,0 29x30), colour toggle: GVL.Diffuse_Sensor_4
        Image (4,4 23x22), image: VisuSymbols.Symbols.RSS1
    Group (1106,177 29x30), colour toggle: GVL.Retroreflective_Sensor_2
        RoundedRectangle (0,0 29x30), colour toggle: GVL.Diffuse_Sensor_4
        Image (4,4 23x22), image: VisuSymbols.Symbols.RSS1
    Group (1105,108 29x30), colour toggle: GVL.Diffuse_Sensor_44
        RoundedRectangle (0,0 29x30), colour toggle: GVL.Diffuse_Sensor_4
        Image (4,4 23x22), image: VisuSymbols.Symbols.RSS1
    Group (1105,241 29x30), colour toggle: GVL.Retroreflective_Sensor_1
        RoundedRectangle (0,0 29x30), colour toggle: GVL.Diffuse_Sensor_4
        Image (4,4 23x22), image: VisuSymbols.Symbols.RSS1
    Group (1105,272 29x30), colour toggle: GVL.Diffuse_Sensor_43
        RoundedRectangle (0,0 29x30), colour toggle: GVL.Diffuse_Sensor_4
        Image (4,4 23x22), image: VisuSymbols.Symbols.RSS1
    Button (478,398 29x30), colour toggle: GVL.Turnable_1_Roll_mas, pressed state: GVL.Turnable_1_Roll_mas
        OnMouseClick: toggle GVL.Turnable_1_Roll_mas
    Image (482,402 23x22), "+", colour toggle: GVL.Turnable_1_Roll_mas, image: VisuSymbols.Symbols.ArrowRoundRightRight
        OnMouseClick: toggle GVL.Turnable_1_Roll_mas
    RoundedRectangle (461,433 29x30), "FL", colour toggle: GVL.Turnable_1_Front_Limit
    Button (511,398 29x30), colour toggle: GVL.Turnable_1_Turn, pressed state: GVL.Turnable_1_Turn
        OnMouseClick: toggle GVL.Turnable_1_Turn
    Image (514,402 23x22), colour toggle: GVL.Turnable_1_Turn, image: VisuSymbols.Symbols.ArrowCircle2LeftUpDown
        OnMouseClick: toggle GVL.Turnable_1_Turn
    Button (544,398 29x30), colour toggle: GVL.Turnable_1_Roll_menos, pressed state: GVL.Turnable_1_Roll_menos
        OnMouseClick: toggle GVL.Turnable_1_Roll_menos
    Image (547,402 23x22), "-", colour toggle: GVL.Turnable_1_Roll_menos, image: VisuSymbols.Symbols.ArrowRoundRightLeft
        OnMouseClick: toggle GVL.Turnable_1_Roll_menos
    RoundedRectangle (494,433 29x30), "BL", colour toggle: GVL.Turnable_1_Back_Limit
    Group (527,433 29x30), colour toggle: GVL.Turnable_1_Limit_90
        RoundedRectangle (0,0 29x30), colour toggle: GVL.Diffuse_Sensor_4
        Image (3,4 23x22), image: VisuSymbols.Symbols.DoubleArrow3
    Group (560,433 29x30), colour toggle: GVL.Turnable_1_Limit_0
        RoundedRectangle (0,0 29x30), colour toggle: GVL.Diffuse_Sensor_4
        Image (4,4 23x22), image: VisuSymbols.Symbols.DoubleArrow4
    RoundedRectangle (852,433 29x30), "FL", colour toggle: GVL.Turnable_1_Front_Limit
    RoundedRectangle (885,433 29x30), "BL", colour toggle: GVL.Turnable_1_Back_Limit
    Group (918,433 29x30), colour toggle: GVL.Turnable_1_Limit_90
        RoundedRectangle (0,0 29x30), colour toggle: GVL.Diffuse_Sensor_4
        Image (3,4 23x22), image: VisuSymbols.Symbols.DoubleArrow3
    Group (951,433 29x30), colour toggle: GVL.Turnable_1_Limit_0
        RoundedRectangle (0,0 29x30), colour toggle: GVL.Diffuse_Sensor_4
        Image (4,4 23x22), image: VisuSymbols.Symbols.DoubleArrow4
    Button (869,398 29x30), colour toggle: GVL.Turnable_2_Roll_mas, pressed state: GVL.Turnable_2_Roll_mas
        OnMouseClick: toggle GVL.Turnable_2_Roll_mas
    Image (873,402 23x22), "+", colour toggle: GVL.Turnable_2_Roll_mas, image: VisuSymbols.Symbols.ArrowRoundRightRight
        OnMouseClick: toggle GVL.Turnable_2_Roll_mas
    Button (902,398 29x30), colour toggle: GVL.Turnable_2_Turn, pressed state: GVL.Turnable_2_Turn
        OnMouseClick: toggle GVL.Turnable_2_Turn
    Image (905,402 23x22), colour toggle: GVL.Turnable_2_Turn, image: VisuSymbols.Symbols.ArrowCircle2LeftUpDown
        OnMouseClick: toggle GVL.Turnable_2_Turn
    Button (935,398 29x30), colour toggle: GVL.Turnable_2_Roll_menos, pressed state: GVL.Turnable_2_Roll_menos
        OnMouseClick: toggle GVL.Turnable_2_Roll_menos
    Image (938,402 23x22), "-", colour toggle: GVL.Turnable_2_Roll_menos, image: VisuSymbols.Symbols.ArrowRoundRightLeft
        OnMouseClick: toggle GVL.Turnable_2_Roll_menos
    Line (1023,226) (1070,258)
    Group (1207,130 29x30), colour toggle: GVL.Stacker_Crane_1_Lift
        OnMouseClick: toggle GVL.Stacker_Crane_1_Lift
        Button (0,0 29x30), colour toggle: GVL.Palletizer_1_Open_Plate, pressed state: GVL.Palletizer_1_Open_Plate
        Image (4,3 22x23), image: VisuSymbols.Symbols.ArrowBoldUp
    Group (1240,129 29x30), colour toggle: GVL.Stacker_Crane_1_Right
        OnMouseClick: toggle GVL.Stacker_Crane_1_Right
        Button (0,0 29x30), colour toggle: GVL.Stacker_Crane_1_Right, pressed state: GVL.Palletizer_1_Open_Plate
            OnMouseClick: toggle GVL.Stacker_Crane_1_Right
        Image (4,4 22x23), image: VisuSymbols.Symbols.ArrowBoldRight
    Group (1275,129 29x30), colour toggle: GVL.Stacker_Crane_1_Left
        OnMouseClick: toggle GVL.Stacker_Crane_1_Left
        Button (0,0 29x30), colour toggle: GVL.Palletizer_1_Open_Plate, pressed state: GVL.Palletizer_1_Open_Plate
        Image (3,4 22x23), image: VisuSymbols.Symbols.ArrowBoldLeft
    Group (1207,164 29x30), colour toggle: GVL.Stacker_Crane_1_Moving_Z
        RoundedRectangle (0,0 29x30), colour toggle: GVL.Diffuse_Sensor_4
        Image (4,4 23x22), image: VisuSymbols.Symbols.DoubleArrow4
    Group (1240,164 29x30), colour toggle: GVL.Stacker_Crane_1_Right_Limit
        RoundedRectangle (0,0 29x30), colour toggle: GVL.Diffuse_Sensor_4
        Image (4,4 23x22), image: VisuSymbols.Symbols.ArrowBoldRight
    Group (1173,164 29x30), colour toggle: GVL.Stacker_Crane_1_Moving_X
        RoundedRectangle (0,0 29x30), colour toggle: GVL.Diffuse_Sensor_4
        Image (3,4 23x22), image: VisuSymbols.Symbols.DoubleArrow3
    Group (1309,164 29x30), colour toggle: GVL.Stacker_Crane_1_Middle_Limit
        RoundedRectangle (0,0 29x30), colour toggle: GVL.Diffuse_Sensor_4
        Image (4,3 22x23), image: VisuSymbols.Symbols.Download
    Group (1275,164 29x30), colour toggle: GVL.Stacker_Crane_1_Left_Limit
        RoundedRectangle (0,0 29x30), colour toggle: GVL.Diffuse_Sensor_4
        Image (3,4 22x23), image: VisuSymbols.Symbols.ArrowBoldLeft
    Rectangle (1899,642 178x262), angle 90
    Rectangle (805,107 29x29), "%i", text variable: GVL.RFID_Reader_1_Command_ID
        p4168582468: GVL.RFID_Reader_1_Command_ID
    Rectangle (776,87 82x16), "Command ID"
    Rectangle (778,142 82x16), "Status"
    Rectangle (778,195 82x16), "Read Data"
    Rectangle (805,161 29x29), "%i", text variable: GVL.RFID_Reader_1_Status
        p4168582468: GVL.RFID_Reader_1_Status
    Rectangle (805,217 29x29), "%i", text variable: GVL.RFID_Reader_1_Read_Data
        p4168582468: GVL.RFID_Reader_1_Read_Data
    PowerSwitch (979,155 35x35), variable: GVL.RFID_Reader_1_Ejecute_Comm, behaviour: TOGGLE, style: Switch-PowerSwitch-Gray
    Rectangle (875,87 82x16), "Command"
    Rectangle (875,142 82x16), "Write Data"
    Rectangle (875,195 82x16), "Memory Index"
    Group (901,107 29x30)
        OnMouseClick: write GVL.RFID_Reader_4_Command_ID via VisuDialogs.Numpad, min 0, max 100, format %i
        Button (0,0 29x30), text variable: GVL.RFID_Reader_1_Command
            OnMouseClick: write GVL.RFID_Reader_4_Command_ID via VisuDialogs.Numpad, min 0, max 100, format %i
        Image (5,5 22x22), image: VisuSymbols.Symbols.Edit
    Group (901,161 29x30)
        OnMouseClick: write GVL.RFID_Reader_4_Write_Data via VisuDialogs.Numpad, min 0, max 100, format %i
        Button (0,0 29x30), text variable: GVL.RFID_Reader_1_Command
            OnMouseClick: write GVL.RFID_Reader_4_Command_ID via VisuDialogs.Numpad, min 0, max 100, format %i
        Image (5,5 22x22), image: VisuSymbols.Symbols.Edit
    Group (901,217 29x30)
        OnMouseClick: write GVL.RFID_Reader_4_Memory_Index via VisuDialogs.Numpad, min 0, max 100, format %i
        Button (0,0 29x30), text variable: GVL.RFID_Reader_1_Command
            OnMouseClick: write GVL.RFID_Reader_4_Command_ID via VisuDialogs.Numpad, min 0, max 100, format %i
        Image (5,5 22x22), image: VisuSymbols.Symbols.Edit
    Rectangle (2440,466 153x409), angle 90
    Rectangle (1421,102 248x30), "Almacén"
    Rectangle (2449,456 103x368), angle 90
    PushSwitch (1487,188 50x50), variable: GVL.Emergency_Stop_9, behaviour: TOGGLE, style: Switch-PushSwitch-Red
    Rectangle (1433,159 177x23), "Emergency Stop"
    Lamp1 (1657,190 50x50), variable: NOT GVL.Safety_Door_13 OR NOT GVL.Safety_Door_14 OR NOT GVL.Safety_Door_15, style: Lamp-Lamp1-Yellow
    Rectangle (1625,159 140x23), "Open_Door"
END_VISUALIZATION

(* stored: Version 1.1.0.1, ProductVersion 3.1.4024.12
   Visu Linea_Almacen_Manual: Id {a071ba1a-b5dd-40c3-94bf-4055c49d6021} *)
